SUBAPPLICATION logiBUS_PI_IDA_OPC (* logiBUS_PI_IDA (Puls-Eingang) auf VT-Zahlenfelder (Zaehler roh + Frequenz Hz, je eigene CNumberVariable) + Bargraph (Frequenz) + OPC-UA (Zaehler DWORD + Frequenz REAL, generisch, ein Kanal) *)
  (* Standard: 61499-2; Description: Copyright (c) 2026 Meisterschulen am Ostbahnhof This program and the accompanying materials are made available under the terms of the Eclipse Public License 2.0 which is available at https://www.eclipse.org/legal/epl-2.0/ SPDX-License-Identifier: EPL-2.0 *)
  (* Version 1.1, 2026-10-03, Franz Höpfinger, Meisterschulen am Ostbahnhof, Folgefix zu FT_DERIV_10_AR v1.2 (K jetzt AUI-Adapter-Socket statt Parameter): bisheriges Parameter Name='K' Value='9' auf FT_DERIV_10_AR entfernt (waere jetzt ein IDE-Fehler, da K kein plain InputVar mehr ist), ersetzt durch LIT_DerivK (initval_AUI, INIT_VAL=9) + AdapterConnection auf FT_DERIV_10_AR.K - gleicher Wert wie bisher, nur adapter-konform verdrahtet. Dieser Baustein hat aktuell keine aktiven Aufrufer im Projekt. *)
  (* Version 1.0, 2026-08-30, Franz Höpfinger, Meisterschulen am Ostbahnhof, initial API and implementation and/or initial documentation *)
  PACKAGE MyLib::sys;
  IMPORT isobus::UT::Q::const::IDs::ID_NULL;
  IMPORT logiBUS::io::PI::logiBUS_PI;
  IMPORT logiBUS::io::PI::logiBUS_PI_S;
  IMPORT logiBUS::utils::conversion::phys::NumericObjectPool_S;
  IMPORT isobus::UT::io::Button::ButtonActivationCode::BT_PRESSED_LATCHED;
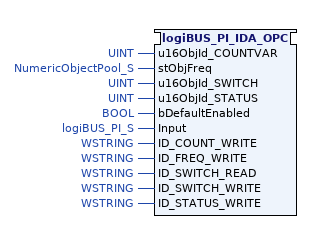
  VAR_INPUT
    u16ObjId_COUNTVAR : UINT := ID_NULL; (* Object ID CNumberVariable (roher Zaehlerstand, unbegrenzt wachsend, Scale=1 im VT-Pool) *)
    stObjFreq : logiBUS::utils::conversion::phys::NumericObjectPool_S := (u16ObjId := ID_NULL, r32Scale := 1.0, i32Offset := 0, u8Decimals := 0); (* Object ID + Scale/Offset/Decimals CNumberVariable (Frequenz Hz, eigene, unabhaengige CNumberVariable - keine Reskalierung des Zaehlers) *)
    u16ObjId_SWITCH : UINT := ID_NULL; (* Object ID Kanal-Ein/Aus-Taste auf der VT (physischer Tastendruck togglet Enable, ueber Button_IE) *)
    u16ObjId_STATUS : UINT := ID_NULL; (* Object ID Status-Anzeige (Hintergrundfarbe Weiss=Kanal deaktiviert / Gruen=aktiv+logiBUS_PI_IDA.QO TRUE / Rot=aktiv+QO FALSE, Stoerung) *)
    bDefaultEnabled : BOOL; (* Kanal-Zustand beim Start: TRUE=aktiv (Kanaele 1-4), FALSE=inaktiv (Kanaele 5-8, da nur 4 Kanaele gleichzeitig verfuegbar sind) *)
    Input : logiBUS::io::PI::logiBUS_PI_S := logiBUS_PI::Invalid; (* Identify the Input PulseInput_I1..I8 *)
    ID_COUNT_WRITE : WSTRING; (* Zaehler-Ruckmelde-Adresse (DWORD, roh, ACTION=PUBLISH) *)
    ID_FREQ_WRITE : WSTRING; (* Frequenz-Ruckmelde-Adresse (REAL Hz, ACTION=PUBLISH) *)
    ID_SWITCH_READ : WSTRING; (* Remote-Schalter-Adresse (BOOL, ACTION=SUBSCRIBE, togglet Kanal-Enable wie ein Tastendruck) *)
    ID_SWITCH_WRITE : WSTRING; (* Echo-Ruckmelde-Adresse (BOOL, ACTION=PUBLISH, aktueller Kanal-Enable-Zustand) *)
    ID_STATUS_WRITE : WSTRING; (* Status-Ruckmelde-Adresse (BOOL, ACTION=PUBLISH, nur lesend, logiBUS_PI_IDA.QO) *)
  END_VAR
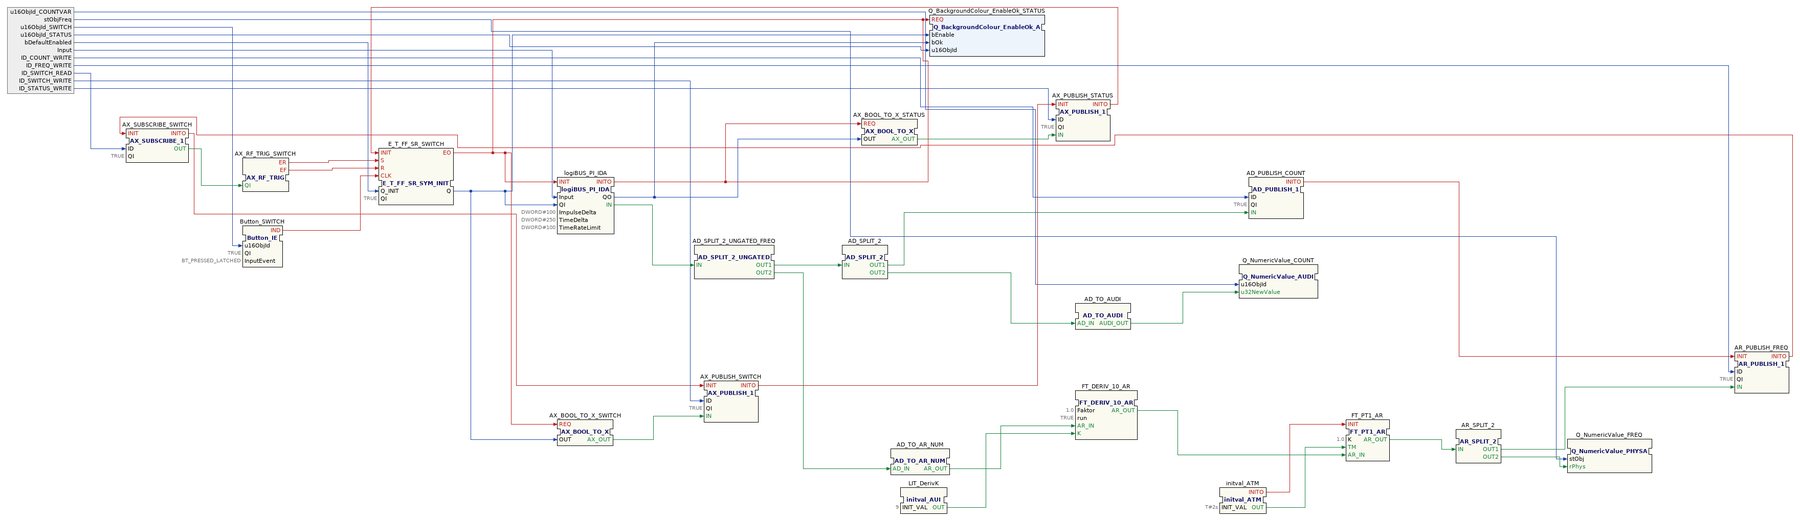
  FBS
    logiBUS_PI_IDA : logiBUS::io::PI::logiBUS_PI_IDA(ImpulseDelta := DWORD#100, TimeDelta := DWORD#250, TimeRateLimit := DWORD#100);
    AD_SPLIT_2_UNGATED_FREQ : adapter::events::unidirectional::AD_SPLIT_2_UNGATED;
    AD_SPLIT_2 : adapter::events::unidirectional::AD_SPLIT_2;
    AD_PUBLISH_COUNT : adapter::net::AD_PUBLISH_1(QI := TRUE);
    AD_TO_AUDI : adapter::conversion::unidirectional::AD_TO_AUDI;
    Q_NumericValue_COUNT : isobus::UT::Q::Q_NumericValue_AUDI;
    AD_TO_AR_NUM : adapter::conversion::unidirectional::AD_TO_AR_NUM;
    AR_PUBLISH_FREQ : adapter::net::AR_PUBLISH_1(QI := TRUE);
    Q_NumericValue_FREQ : isobus::UT::Q::Q_NumericValue_PHYSA;
    AR_SPLIT_2 : adapter::events::unidirectional::AR_SPLIT_2;
    E_T_FF_SR_SWITCH : iec61499::events::E_T_FF_SR_SYM_INIT(QI := TRUE);
    Button_SWITCH : isobus::UT::io::Button::Button_IE(QI := TRUE, InputEvent := BT_PRESSED_LATCHED);
    AX_SUBSCRIBE_SWITCH : adapter::net::AX_SUBSCRIBE_1(QI := TRUE);
    AX_RF_TRIG_SWITCH : adapter::events::unidirectional::AX_RF_TRIG;
    AX_BOOL_TO_X_SWITCH : adapter::conversion::unidirectional::AX_BOOL_TO_X;
    AX_PUBLISH_SWITCH : adapter::net::AX_PUBLISH_1(QI := TRUE);
    AX_BOOL_TO_X_STATUS : adapter::conversion::unidirectional::AX_BOOL_TO_X;
    AX_PUBLISH_STATUS : adapter::net::AX_PUBLISH_1(QI := TRUE);
    initval_ATM : adapter::types::unidirectional::ATM::initval::initval_ATM(INIT_VAL := T#2s);
    FT_PT1_AR : OSCAT_adapter::Control::FT_PT1_AR(K := 1.0);
    FT_DERIV_10_AR : OSCAT_adapter::Control::FT_DERIV_10_AR(Faktor := 1.0, run := TRUE);
    LIT_DerivK : adapter::types::unidirectional::AUI::initval::initval_AUI(INIT_VAL := 9);
  END_FBS
  SUBAPPS
    Q_BackgroundColour_EnableOk_STATUS : MyLib::sys::Q_BackgroundColour_EnableOk_A;
  END_SUBAPPS
  EVENT_CONNECTIONS
    AD_PUBLISH_COUNT.INITO TO AR_PUBLISH_FREQ.INIT;
    AR_PUBLISH_FREQ.INITO TO AX_SUBSCRIBE_SWITCH.INIT;
    AX_SUBSCRIBE_SWITCH.INITO TO AX_PUBLISH_SWITCH.INIT;
    AX_PUBLISH_SWITCH.INITO TO AX_PUBLISH_STATUS.INIT;
    AX_PUBLISH_STATUS.INITO TO E_T_FF_SR_SWITCH.INIT;
    E_T_FF_SR_SWITCH.EO TO logiBUS_PI_IDA.INIT;
    E_T_FF_SR_SWITCH.EO TO Q_BackgroundColour_EnableOk_STATUS.REQ;
    logiBUS_PI_IDA.INITO TO Q_BackgroundColour_EnableOk_STATUS.REQ;
    logiBUS_PI_IDA.INITO TO AX_BOOL_TO_X_STATUS.REQ;
    AX_RF_TRIG_SWITCH.ER TO E_T_FF_SR_SWITCH.S;
    AX_RF_TRIG_SWITCH.EF TO E_T_FF_SR_SWITCH.R;
    Button_SWITCH.IND TO E_T_FF_SR_SWITCH.CLK;
    E_T_FF_SR_SWITCH.EO TO AX_BOOL_TO_X_SWITCH.REQ;
    initval_ATM.INITO TO FT_PT1_AR.INIT;
  END_CONNECTIONS
  DATA_CONNECTIONS
    Input TO logiBUS_PI_IDA.Input;
    u16ObjId_COUNTVAR TO Q_NumericValue_COUNT.u16ObjId;
    stObjFreq TO Q_NumericValue_FREQ.stObj;
    ID_COUNT_WRITE TO AD_PUBLISH_COUNT.ID;
    ID_FREQ_WRITE TO AR_PUBLISH_FREQ.ID;
    bDefaultEnabled TO E_T_FF_SR_SWITCH.Q_INIT;
    E_T_FF_SR_SWITCH.Q TO logiBUS_PI_IDA.QI;
    E_T_FF_SR_SWITCH.Q TO Q_BackgroundColour_EnableOk_STATUS.bEnable;
    logiBUS_PI_IDA.QO TO Q_BackgroundColour_EnableOk_STATUS.bOk;
    u16ObjId_STATUS TO Q_BackgroundColour_EnableOk_STATUS.u16ObjId;
    E_T_FF_SR_SWITCH.Q TO AX_BOOL_TO_X_SWITCH.OUT;
    logiBUS_PI_IDA.QO TO AX_BOOL_TO_X_STATUS.OUT;
    ID_SWITCH_READ TO AX_SUBSCRIBE_SWITCH.ID;
    ID_SWITCH_WRITE TO AX_PUBLISH_SWITCH.ID;
    ID_STATUS_WRITE TO AX_PUBLISH_STATUS.ID;
    u16ObjId_SWITCH TO Button_SWITCH.u16ObjId;
  END_CONNECTIONS
  ADAPTER_CONNECTIONS
    logiBUS_PI_IDA.IN TO AD_SPLIT_2_UNGATED_FREQ.IN;
    AD_SPLIT_2_UNGATED_FREQ.OUT1 TO AD_SPLIT_2.IN;
    AD_SPLIT_2_UNGATED_FREQ.OUT2 TO AD_TO_AR_NUM.AD_IN;
    AD_SPLIT_2.OUT1 TO AD_PUBLISH_COUNT.IN;
    AD_SPLIT_2.OUT2 TO AD_TO_AUDI.AD_IN;
    AD_TO_AUDI.AUDI_OUT TO Q_NumericValue_COUNT.u32NewValue;
    AR_SPLIT_2.OUT1 TO AR_PUBLISH_FREQ.IN;
    AR_SPLIT_2.OUT2 TO Q_NumericValue_FREQ.rPhys;
    AX_SUBSCRIBE_SWITCH.OUT TO AX_RF_TRIG_SWITCH.QI;
    AX_BOOL_TO_X_SWITCH.AX_OUT TO AX_PUBLISH_SWITCH.IN;
    AX_BOOL_TO_X_STATUS.AX_OUT TO AX_PUBLISH_STATUS.IN;
    initval_ATM.OUT TO FT_PT1_AR.TM;
    FT_DERIV_10_AR.AR_OUT TO FT_PT1_AR.AR_IN;
    AD_TO_AR_NUM.AR_OUT TO FT_DERIV_10_AR.AR_IN;
    LIT_DerivK.OUT TO FT_DERIV_10_AR.K;
    FT_PT1_AR.AR_OUT TO AR_SPLIT_2.IN;
  END_CONNECTIONS
END_SUBAPPLICATION
